FUNCTION_BLOCK FB_RealControlBox IMPLEMENTS I_CraneControlBox
VAR_INPUT
END_VAR
VAR_OUTPUT
END_VAR
VAR
END_VAR

{warning 'add method implementation '}
METHOD Joystick : REAL
Joystick := 0.0;
END_METHOD

{warning 'add method implementation '}
METHOD Mode : E_ControlBoxSwitchMode
Mode := E_ControlBoxSwitchMode.Off;
END_METHOD

{warning 'add method implementation '}
METHOD Status : E_RunningStates
Status := E_RunningStates.NotReady;
END_METHOD

END_FUNCTION_BLOCK

(* stored: Version 1.1.0.1, ProductVersion 3.1.4024.12
   POU FB_RealControlBox: Id {e760bdee-97ca-4a12-b73e-bf247f0f3ce6}, SpecialFunc None
   Method Joystick: Id {7024017e-12eb-4310-b9bb-d769ee14219e}
   Method Mode: Id {124a7371-d47b-4744-bcbe-99bdc418ae05}
   Method Status: Id {dffca296-d0eb-401b-a9eb-bfd24e35a824} *)
